(* CoDeSys 2.3.9.47 project: 1floor_2016_06_22_beta.pr6 *)
(* Libraries: TcBABasicBC.lb6 22.7.15 15:46:36, TcPlcUtilitiesBC.lb6 13.5.05 11:19:40, PlcSystemBC.lb6 21.3.01 11:03:02, TcAdsBC.lb6 5.7.02 11:03:02, standard.lb6 5.6.98 11:03:02 *)

(* Global variable list: main *)
VAR_GLOBAL


(*ADS*)

	ads_adr1: STRING:='10.0.5.61.1.1';
	ads_adr2: STRING:='10.0.5.62.1.1';
	ads_adr3: STRING:='10.0.5.63.1.1';

	write_ads: ADSWRITE;

	data2floor: ARRAY[0..3] OF BYTE;
	data2floor_prev :ARRAY[0..3] OF BYTE;
	data3floor: ARRAY[0..10] OF BYTE;
	data3floor_prev :ARRAY[0..10] OF BYTE;

	m_fancoil_vitalnya_low 			AT%MX300.0: BOOL;
	m_fancoil_vitalnya_med 			AT%MX300.1: BOOL;
	m_fancoil_vitalnya_high 			AT%MX300.2: BOOL;
	skvazhyna 						AT%MX300.3:BOOL;
	tepla_pidloga					AT%MX300.4:BOOL;

	T_out3							AT%MB303:BYTE;


	iHour							AT%MB304:BYTE;
	iMinute							AT%MB305:BYTE;
	lights							AT%MB306:DWORD;

	sw_tambur2_1					AT%MX200.0:BOOL;
	sw_tambur3_2					AT%MX300.1:BOOL;
	bDarkOutside					AT%MX300.6:BOOL;
	bT_out_sign						AT%MX300.7:BOOL;

	eib_komora_l 					AT%MX400.0:BOOL;
	eib_su1_l 						AT%MX400.1:BOOL;
	eib_topochna_l 					AT%MX400.2:BOOL;
	eib_su2_bra	 					AT%MX400.3:BOOL;
	eib_su2_l 						AT%MX400.4:BOOL;
	eib_su1_rakovyna 				AT%MX400.5:BOOL;
	eib_su2_dush 					AT%MX400.6:BOOL;
	eib_dush 						AT%MX400.7:BOOL;

	eib_kuhnya1	 				AT%MX401.0:BOOL;
	eib_vitalnya_smugy1 			AT%MX401.1:BOOL;
	eib_vitalnya_l 					AT%MX401.2:BOOL;
	eib_vitalnya_prokladka 			AT%MX401.3:BOOL;
	eib_terassa_stina	 			AT%MX401.4:BOOL;
	eib_pidval_shody	 			AT%MX401.5:BOOL;
	eib_skhody2pov 				AT%MX401.6:BOOL;
	eib_tambur_l 					AT%MX401.7:BOOL;

	eib_vent_su1 					AT%MX402.0:BOOL;
	eib_vent_kuh_low 				AT%MX402.1:BOOL;
	eib_vent_dush 					AT%MX402.2:BOOL;
	eib_vent_komora 				AT%MX402.3:BOOL;
	eib_vent_kuh_high 				AT%MX403.4:BOOL;

END_VAR

(* Global variable list: physical *)
VAR_GLOBAL



	moove_su1				AT %IX80.0:	BOOL;
	moove_topochna			AT %IX80.1:	BOOL;
	moove_su2				AT %IX80.2:	BOOL;
	moove_korydor_ops		AT %IX80.3:	BOOL;
	moove_korydor			AT %IX80.4:	BOOL;
	moove_vitalnya			AT %IX80.5:	BOOL;
	moove_komora			AT %IX80.6:	BOOL;
(*	din1_8	AT %IX80.7:	BOOL;*)
	moove_kino				AT %IX81.0:	BOOL;
	moove_skhody2_3		AT %IX81.1:	BOOL;
	moove_skhody1_2		AT %IX81.2:	BOOL;
	moove_garderob			AT %IX81.3:	BOOL;
	moove_studio			AT %IX81.4:	BOOL;
	moove_tambur3			AT %IX81.5:	BOOL;
	moove_kabinet			AT %IX81.6:	BOOL;
	moove_dytjacha			AT %IX81.7:	BOOL;
	moove_spalnya			AT %IX82.0:	BOOL;
(*	din3_2	AT %IX82.1:	BOOL;*)
	moove_korydor3			AT %IX82.2:	BOOL;
(*	din3_4	AT %IX82.3:	BOOL;
	din3_5	AT %IX82.4:	BOOL;
	din3_6	AT %IX82.5:	BOOL;
	din3_7	AT %IX82.6:	BOOL;
	din3_8sw_vhid2		AT %IX82.7:	BOOL;
	din4_1	AT %IX83.0:	BOOL;
*)
	sw_su1_2				AT %IX83.1:	BOOL;
	sw_komora1				AT %IX83.2:	BOOL;
	sw_vhid1					AT %IX83.3:	BOOL;
	sw_topochna2			AT %IX83.4:	BOOL;
	sw_vhid2					AT %IX83.5:	BOOL;
	sw_topochna1			AT %IX83.6:	BOOL;
	sw_su1_1				AT %IX83.7:	BOOL;
	sw_tambur1_2			AT %IX84.0:	BOOL;
	sw_su2					AT %IX84.1:	BOOL;
	sw_kuh_su2				AT %IX84.2:	BOOL;
	sw_kuh3					AT %IX84.3:	BOOL;
(*	din5_5	AT %IX84.4:	BOOL;*)
	sw_kuh4					AT %IX84.5:	BOOL;
	sw_tambur1				AT %IX84.6:	BOOL;
	sw_vitalnya1				AT %IX84.7:	BOOL;
	sw_vitalnya2				AT %IX85.0:	BOOL;
	sw_kuh2					AT %IX85.1:	BOOL;
(*	din6_3	AT %IX85.2:	BOOL;*)
	sw_kuh1					AT %IX85.3:	BOOL;
	sw_vitalnya3				AT %IX85.4:	BOOL;
	sw_tambur3				AT %IX85.5:	BOOL;
	sw_tambur_su			AT %IX85.6:	BOOL;
	sw_transit2pov			AT %IX85.7:	BOOL;

	ch_sensor1				AT %IX86.0:	BOOL;
	ch_sensor2				AT %IX86.1:	BOOL;
	zatoplennya_kot			AT %IX86.2:	BOOL;
	zatoplennya_komora		AT %IX86.3:	BOOL;
	zatoplennya_su2			AT %IX86.4:	BOOL;
	zatoplennya_kuh			AT %IX86.5:	BOOL;
	zatoplennya_su3pov		AT %IX86.6:	BOOL;
(*	din7_8	AT %IX86.7:	BOOL;*)

	komora_l				AT %QX80.0:	BOOL;
	su1_l					AT %QX80.1:	BOOL;
	topochna_l				AT %QX80.2:	BOOL;
	su2_bra					AT %QX80.3:	BOOL;
	topochna2_l				AT %QX80.4:	BOOL;
	su2_l					AT %QX80.5:	BOOL;
	su1_rakovyna			AT %QX80.6:	BOOL;
	su2_dush				AT %QX80.7:	BOOL;
	dush					AT %QX81.0:	BOOL;
	vitalnya_smugy2			AT %QX81.1:	BOOL;
	su2_polytsi				AT %QX81.2:	BOOL;
	fancoil_vitalnya_low		AT %QX81.3:	BOOL;
	kuhnya1					AT %QX81.4:	BOOL;
	fancoil_vitalnya_med		AT %QX81.5:	BOOL;
	kuhnya2					AT %QX81.6:	BOOL;
	fancoil_vitalnya_high		AT %QX81.7:	BOOL;
	w_valve_recirc			AT %QX82.0:	BOOL;
(*	dout3_2	AT %QX82.1:	BOOL;*)
	w_valve3pov				AT %QX82.2:	BOOL;
	vitalnya_smugy1			AT %QX82.3:	BOOL;
	w_valve1pov				AT %QX82.4:	BOOL;
	vitalnya_l				AT %QX82.5:	BOOL;
	freecooling				AT %QX82.6:	BOOL;
	vitalnya_prokladka		AT %QX82.7:	BOOL;
	terassa_stina				AT %QX83.0:	BOOL;
	pidval_shody				AT %QX83.1:	BOOL;
	terassa					AT %QX83.2:	BOOL;
	skhody2pov				AT %QX83.3:	BOOL;
(*	dout4_5	AT %QX83.4:	BOOL;
	dout4_6	AT %QX83.5:	BOOL;
*)	dout4_7	AT %QX83.6:	BOOL;

	tambur_l					AT %QX83.7:	BOOL;
(*	dout5_1	AT %QX84.0:	BOOL;
	dout5_2 AT %QX84.1:	BOOL;
*)	gas_valve				AT %QX84.2:	BOOL;
(*	dout5_4	AT %QX84.3:	BOOL;
	dout5_5	AT %QX84.4:	BOOL;
	dout5_6	AT %QX84.5:	BOOL;
	dout5_7	AT %QX84.6:	BOOL;
	dout5_8	AT %QX84.7:	BOOL;
	dout6_1	AT %QX85.0:	BOOL;
	dout6_2	AT %QX85.1:	BOOL;
	dout6_3	AT %QX85.2:	BOOL;
	dout6_4	AT %QX85.3:	BOOL;
	dout6_5	AT %QX85.4:	BOOL;
	dout6_6	AT %QX85.5:	BOOL;
	dout6_7	AT %QX85.6:	BOOL;
	dout6_8	AT %QX85.7:	BOOL;
	dout7_1	AT %QX86.0:	BOOL;
	dout7_2	AT %QX86.1:	BOOL;
	dout7_3	AT %QX86.2:	BOOL;
	dout7_4	AT %QX86.3:	BOOL;
	dout7_5	AT %QX86.4:	BOOL;
	dout7_6	AT %QX86.5:	BOOL;
	dout7_7	AT %QX86.6:	BOOL;
	dout7_8	AT %QX86.7:	BOOL;
	dout8_1	AT %QX87.0:	BOOL;
	dout8_2	AT %QX87.1:	BOOL;
	dout8_3	AT %QX87.2:	BOOL;
	dout8_4	AT %QX87.3:	BOOL;
	dout8_5	AT %QX87.4:	BOOL;
	dout8_6	AT %QX87.5:	BOOL;
	dout8_7	AT %QX87.6:	BOOL;
	dout8_8	AT %QX87.7:	BOOL;
*)	vent_su1					AT %QX88.0:	BOOL;
	vent_kuh_low				AT %QX88.1:	BOOL;
	vent_dush				AT %QX88.2:	BOOL;
	collector_komora			AT %QX88.3:	BOOL;
	vent_komora				AT %QX88.4:	BOOL;
	collector_kuh				AT %QX88.5:	BOOL;
	vent_kuh_high			AT %QX88.6:	BOOL;
	collector_vitalnya1			AT %QX88.7:	BOOL;
	collector_vitalnya2			AT %QX89.0:	BOOL;
(*	dout10_2	AT %QX89.1:	BOOL;
*)	collector_su2				AT %QX89.2:	BOOL;
(*	dout10_4	AT %QX89.3:	BOOL;
*)	collector_vhid_stina		AT %QX89.4:	BOOL;
(*	dout10_6	AT %QX89.5:	BOOL;
*)	collector_vhid				AT %QX89.6:	BOOL;
(*	dout10_8	AT %QX89.7:	BOOL;
	dout11_1	AT %QX90.0:	BOOL;
	dout11_2	AT %QX90.1:	BOOL;
	dout11_3	AT %QX90.2:	BOOL;
	dout11_4	AT %QX90.3:	BOOL;
	dout11_5	AT %QX90.4:	BOOL;
	dout11_6	AT %QX90.5:	BOOL;
	dout11_7	AT %QX90.6:	BOOL;
	dout11_8	AT %QX90.7:	BOOL;
*)
	klapan_vitalnya			AT %QB2:	INT;
	KL4414_2_Out			AT %QB6:	INT;
	KL4414_3_Out			AT %QB10:	INT;
	KL4414_4_Out			AT %QB14:	INT;

	temp_vhid	AT %IB50:	INT; (*25*)
	temp_dush	AT %IB58:	INT;(*25*)
	temp_kuh	AT %IB66:	INT;(*-136*)
	temp_vhid_stina	AT %IB70:	INT;(*0*)
(*
(* @GLOBAL_VARIABLE_LIST := TwinCAT_Import *)
(* @PATH := '' *)
VAR_GLOBAL (* DO NOT CHANGE THIS SHEET MANUALLY! *)
	PlcInVar_0	AT %QB128:	USINT;
	PlcInVar_1	AT %QB129:	USINT;
	PlcInVar_2	AT %QB130:	USINT;
	PlcInVar_3	AT %QB131:	USINT;
	PlcInVar_4	AT %QB132:	USINT;
	PlcInVar_5	AT %QB133:	USINT;
	PlcInVar_6	AT %QB134:	USINT;
	PlcInVar_7	AT %QB135:	USINT;
	PlcInVar_8	AT %QB136:	USINT;
	PlcInVar_9	AT %QB137:	USINT;
	PlcInVar_10	AT %QB138:	USINT;
	PlcInVar_11	AT %QB139:	USINT;
	PlcInVar_12	AT %QB140:	USINT;
	PlcInVar_13	AT %QB141:	USINT;
	PlcInVar_14	AT %QB142:	USINT;
	PlcInVar_15	AT %QB143:	USINT;
	PlcOutVar_0	AT %IB128:	USINT;
	PlcOutVar_1	AT %IB129:	USINT;
	PlcOutVar_2	AT %IB130:	USINT;
	PlcOutVar_3	AT %IB131:	USINT;
	PlcOutVar_4	AT %IB132:	USINT;
	PlcOutVar_5	AT %IB133:	USINT;
	PlcOutVar_6	AT %IB134:	USINT;
	PlcOutVar_7	AT %IB135:	USINT;
	PlcOutVar_8	AT %IB136:	USINT;
	PlcOutVar_9	AT %IB137:	USINT;
	PlcOutVar_10	AT %IB138:	USINT;
	PlcOutVar_11	AT %IB139:	USINT;
	PlcOutVar_12	AT %IB140:	USINT;
	PlcOutVar_13	AT %IB141:	USINT;
	PlcOutVar_14	AT %IB142:	USINT;
	PlcOutVar_15	AT %IB143:	USINT;
	Term_2_KL4414_1_State	AT %IB0:	USINT;
	Term_2_KL4414_1_Data_In	AT %IB2:	INT;
	Term_2_KL4414_1_Ctrl	AT %QB0:	USINT;
	Term_2_KL4414_1_Data_Out	AT %QB2:	INT;
	Term_2_KL4414_2_State	AT %IB4:	USINT;
	Term_2_KL4414_2_Data_In	AT %IB6:	INT;
	Term_2_KL4414_2_Ctrl	AT %QB4:	USINT;
	Term_2_KL4414_2_Data_Out	AT %QB6:	INT;
	Term_2_KL4414_3_State	AT %IB8:	USINT;
	Term_2_KL4414_3_Data_In	AT %IB10:	INT;
	Term_2_KL4414_3_Ctrl	AT %QB8:	USINT;
	Term_2_KL4414_3_Data_Out	AT %QB10:	INT;
	Term_2_KL4414_4_State	AT %IB12:	USINT;
	Term_2_KL4414_4_Data_In	AT %IB14:	INT;
	Term_2_KL4414_4_Ctrl	AT %QB12:	USINT;
	Term_2_KL4414_4_Data_Out	AT %QB14:	INT;
	Term_14_KL3228_4_1_State	AT %IB16:	USINT;
	Term_14_KL3228_4_1_Data_In	AT %IB18:	INT;
	Term_14_KL3228_4_1_Ctrl	AT %QB16:	USINT;
	Term_14_KL3228_4_1_Data_Out	AT %QB18:	INT;
	Term_14_KL3228_4_2_State	AT %IB20:	USINT;
	Term_14_KL3228_4_2_Data_In	AT %IB22:	INT;
	Term_14_KL3228_4_2_Ctrl	AT %QB20:	USINT;
	Term_14_KL3228_4_2_Data_Out	AT %QB22:	INT;
	Term_14_KL3228_4_3_State	AT %IB24:	USINT;
	Term_14_KL3228_4_3_Data_In	AT %IB26:	INT;
	Term_14_KL3228_4_3_Ctrl	AT %QB24:	USINT;
	Term_14_KL3228_4_3_Data_Out	AT %QB26:	INT;
	Term_14_KL3228_4_4_State	AT %IB28:	USINT;
	Term_14_KL3228_4_4_Data_In	AT %IB30:	INT;
	Term_14_KL3228_4_4_Ctrl	AT %QB28:	USINT;
	Term_14_KL3228_4_4_Data_Out	AT %QB30:	INT;
	Term_15_KL3228_4_1_State	AT %IB32:	USINT;
	Term_15_KL3228_4_1_Data_In	AT %IB34:	INT;
	Term_15_KL3228_4_1_Ctrl	AT %QB32:	USINT;
	Term_15_KL3228_4_1_Data_Out	AT %QB34:	INT;
	Term_15_KL3228_4_2_State	AT %IB36:	USINT;
	Term_15_KL3228_4_2_Data_In	AT %IB38:	INT;
	Term_15_KL3228_4_2_Ctrl	AT %QB36:	USINT;
	Term_15_KL3228_4_2_Data_Out	AT %QB38:	INT;
	Term_15_KL3228_4_3_State	AT %IB40:	USINT;
	Term_15_KL3228_4_3_Data_In	AT %IB42:	INT;
	Term_15_KL3228_4_3_Ctrl	AT %QB40:	USINT;
	Term_15_KL3228_4_3_Data_Out	AT %QB42:	INT;
	Term_15_KL3228_4_4_State	AT %IB44:	USINT;
	Term_15_KL3228_4_4_Data_In	AT %IB46:	INT;
	Term_15_KL3228_4_4_Ctrl	AT %QB44:	USINT;
	Term_15_KL3228_4_4_Data_Out	AT %QB46:	INT;
	Term_16_KL3228_4_1_State	AT %IB48:	USINT;
	Term_16_KL3228_4_1_Data_In	AT %IB50:	INT;
	Term_16_KL3228_4_1_Ctrl	AT %QB48:	USINT;
	Term_16_KL3228_4_1_Data_Out	AT %QB50:	INT;
	Term_16_KL3228_4_2_State	AT %IB52:	USINT;
	Term_16_KL3228_4_2_Data_In	AT %IB54:	INT;
	Term_16_KL3228_4_2_Ctrl	AT %QB52:	USINT;
	Term_16_KL3228_4_2_Data_Out	AT %QB54:	INT;
	Term_16_KL3228_4_3_State	AT %IB56:	USINT;
	Term_16_KL3228_4_3_Data_In	AT %IB58:	INT;
	Term_16_KL3228_4_3_Ctrl	AT %QB56:	USINT;
	Term_16_KL3228_4_3_Data_Out	AT %QB58:	INT;
	Term_16_KL3228_4_4_State	AT %IB60:	USINT;
	Term_16_KL3228_4_4_Data_In	AT %IB62:	INT;
	Term_16_KL3228_4_4_Ctrl	AT %QB60:	USINT;
	Term_16_KL3228_4_4_Data_Out	AT %QB62:	INT;
	Term_17_KL3228_4_1_State	AT %IB64:	USINT;
	Term_17_KL3228_4_1_Data_In	AT %IB66:	INT;
	Term_17_KL3228_4_1_Ctrl	AT %QB64:	USINT;
	Term_17_KL3228_4_1_Data_Out	AT %QB66:	INT;
	Term_17_KL3228_4_2_State	AT %IB68:	USINT;
	Term_17_KL3228_4_2_Data_In	AT %IB70:	INT;
	Term_17_KL3228_4_2_Ctrl	AT %QB68:	USINT;
	Term_17_KL3228_4_2_Data_Out	AT %QB70:	INT;
	Term_17_KL3228_4_3_State	AT %IB72:	USINT;
	Term_17_KL3228_4_3_Data_In	AT %IB74:	INT;
	Term_17_KL3228_4_3_Ctrl	AT %QB72:	USINT;
	Term_17_KL3228_4_3_Data_Out	AT %QB74:	INT;
	Term_17_KL3228_4_4_State	AT %IB76:	USINT;
	Term_17_KL3228_4_4_Data_In	AT %IB78:	INT;
	Term_17_KL3228_4_4_Ctrl	AT %QB76:	USINT;
	Term_17_KL3228_4_4_Data_Out	AT %QB78:	INT; 
	Term_3_KL2408_1_Output	AT %QX80.0:	BOOL;
	Term_3_KL2408_2_Output	AT %QX80.1:	BOOL;
	Term_3_KL2408_3_Output	AT %QX80.2:	BOOL;
	Term_3_KL2408_4_Output	AT %QX80.3:	BOOL;
	Term_3_KL2408_5_Output	AT %QX80.4:	BOOL;
	Term_3_KL2408_6_Output	AT %QX80.5:	BOOL;
	Term_3_KL2408_7_Output	AT %QX80.6:	BOOL;
	Term_3_KL2408_8_Output	AT %QX80.7:	BOOL;
	Term_4_KL2408_1_Output	AT %QX81.0:	BOOL;
	Term_4_KL2408_2_Output	AT %QX81.1:	BOOL;
	Term_4_KL2408_3_Output	AT %QX81.2:	BOOL;
	Term_4_KL2408_4_Output	AT %QX81.3:	BOOL;
	Term_4_KL2408_5_Output	AT %QX81.4:	BOOL;
	Term_4_KL2408_6_Output	AT %QX81.5:	BOOL;
	Term_4_KL2408_7_Output	AT %QX81.6:	BOOL;
	Term_4_KL2408_8_Output	AT %QX81.7:	BOOL;
	Term_5_KL2408_1_Output	AT %QX82.0:	BOOL;
	Term_5_KL2408_2_Output	AT %QX82.1:	BOOL;
	Term_5_KL2408_3_Output	AT %QX82.2:	BOOL;
	Term_5_KL2408_4_Output	AT %QX82.3:	BOOL;
	Term_5_KL2408_5_Output	AT %QX82.4:	BOOL;
	Term_5_KL2408_6_Output	AT %QX82.5:	BOOL;
	Term_5_KL2408_7_Output	AT %QX82.6:	BOOL;
	Term_5_KL2408_8_Output	AT %QX82.7:	BOOL;
	Term_6_KL2408_1_Output	AT %QX83.0:	BOOL;
	Term_6_KL2408_2_Output	AT %QX83.1:	BOOL;
	Term_6_KL2408_3_Output	AT %QX83.2:	BOOL;
	Term_6_KL2408_4_Output	AT %QX83.3:	BOOL;
	Term_6_KL2408_5_Output	AT %QX83.4:	BOOL;
	Term_6_KL2408_6_Output	AT %QX83.5:	BOOL;
	Term_6_KL2408_7_Output	AT %QX83.6:	BOOL;
	Term_6_KL2408_8_Output	AT %QX83.7:	BOOL;
	Term_7_KL2408_1_Output	AT %QX84.0:	BOOL;
	Term_7_KL2408_2_Output	AT %QX84.1:	BOOL;
	Term_7_KL2408_3_Output	AT %QX84.2:	BOOL;
	Term_7_KL2408_4_Output	AT %QX84.3:	BOOL;
	Term_7_KL2408_5_Output	AT %QX84.4:	BOOL;
	Term_7_KL2408_6_Output	AT %QX84.5:	BOOL;
	Term_7_KL2408_7_Output	AT %QX84.6:	BOOL;
	Term_7_KL2408_8_Output	AT %QX84.7:	BOOL;
	Term_8_KL2408_1_Output	AT %QX85.0:	BOOL;
	Term_8_KL2408_2_Output	AT %QX85.1:	BOOL;
	Term_8_KL2408_3_Output	AT %QX85.2:	BOOL;
	Term_8_KL2408_4_Output	AT %QX85.3:	BOOL;
	Term_8_KL2408_5_Output	AT %QX85.4:	BOOL;
	Term_8_KL2408_6_Output	AT %QX85.5:	BOOL;
	Term_8_KL2408_7_Output	AT %QX85.6:	BOOL;
	Term_8_KL2408_8_Output	AT %QX85.7:	BOOL;
	Term_9_KL2408_1_Output	AT %QX86.0:	BOOL;
	Term_9_KL2408_2_Output	AT %QX86.1:	BOOL;
	Term_9_KL2408_3_Output	AT %QX86.2:	BOOL;
	Term_9_KL2408_4_Output	AT %QX86.3:	BOOL;
	Term_9_KL2408_5_Output	AT %QX86.4:	BOOL;
	Term_9_KL2408_6_Output	AT %QX86.5:	BOOL;
	Term_9_KL2408_7_Output	AT %QX86.6:	BOOL;
	Term_9_KL2408_8_Output	AT %QX86.7:	BOOL;
	Term_10_KL2408_1_Output	AT %QX87.0:	BOOL;
	Term_10_KL2408_2_Output	AT %QX87.1:	BOOL;
	Term_10_KL2408_3_Output	AT %QX87.2:	BOOL;
	Term_10_KL2408_4_Output	AT %QX87.3:	BOOL;
	Term_10_KL2408_5_Output	AT %QX87.4:	BOOL;
	Term_10_KL2408_6_Output	AT %QX87.5:	BOOL;
	Term_10_KL2408_7_Output	AT %QX87.6:	BOOL;
	Term_10_KL2408_8_Output	AT %QX87.7:	BOOL;
	Term_11_KL2408_1_Output	AT %QX88.0:	BOOL;
	Term_11_KL2408_2_Output	AT %QX88.1:	BOOL;
	Term_11_KL2408_3_Output	AT %QX88.2:	BOOL;
	Term_11_KL2408_4_Output	AT %QX88.3:	BOOL;
	Term_11_KL2408_5_Output	AT %QX88.4:	BOOL;
	Term_11_KL2408_6_Output	AT %QX88.5:	BOOL;
	Term_11_KL2408_7_Output	AT %QX88.6:	BOOL;
	Term_11_KL2408_8_Output	AT %QX88.7:	BOOL;
	Term_12_KL2408_1_Output	AT %QX89.0:	BOOL;
	Term_12_KL2408_2_Output	AT %QX89.1:	BOOL;
	Term_12_KL2408_3_Output	AT %QX89.2:	BOOL;
	Term_12_KL2408_4_Output	AT %QX89.3:	BOOL;
	Term_12_KL2408_5_Output	AT %QX89.4:	BOOL;
	Term_12_KL2408_6_Output	AT %QX89.5:	BOOL;
	Term_12_KL2408_7_Output	AT %QX89.6:	BOOL;
	Term_12_KL2408_8_Output	AT %QX89.7:	BOOL;
	Term_13_KL2408_1_Output	AT %QX90.0:	BOOL;
	Term_13_KL2408_2_Output	AT %QX90.1:	BOOL;
	Term_13_KL2408_3_Output	AT %QX90.2:	BOOL;
	Term_13_KL2408_4_Output	AT %QX90.3:	BOOL;
	Term_13_KL2408_5_Output	AT %QX90.4:	BOOL;
	Term_13_KL2408_6_Output	AT %QX90.5:	BOOL;
	Term_13_KL2408_7_Output	AT %QX90.6:	BOOL;
	Term_13_KL2408_8_Output	AT %QX90.7:	BOOL;
	
END_VAR

*)
END_VAR

(* Data type *)
TYPE ContactType: (NO,NC);
(*NO - sensor sends TRUE on triggering and FALSE in normal state.
NC - sensor sends FALSE on triggering and TRUE in normal state *)

END_TYPE

(* Data type *)
TYPE   ManSwitch: (OFF, ON, AUTO);
END_TYPE

(* Data type *)
TYPE ROOM_HVAC :
STRUCT

	heat_mode:STRING;
	heat_speed:USINT;

	delta_t:SINT;
	t_cur:SINT;
	t_ust:SINT;

	fancoil_speed:SINT;
	klapan:WORD;

	collector1: BOOL;
	collector2: BOOL;
	collector3: BOOL;
	collector4: BOOL;

END_STRUCT
END_TYPE

(* Data type *)
TYPE WaterLeakageDetectionCfg :
	STRUCT
		sensorContacts:ContactType:=NO;
		valveContacts:ContactType:=NO;
		sensorDelay:TIME:=t#5s;
		waterOnTimerDelay: TIME:=t#10ms;
	END_STRUCT
END_TYPE

(* POU MAIN, ST *)
PROGRAM MAIN
VAR

	i:INT;
END_VAR
WaterAndGasLeakage;
Light;
heat;
ADS_write;
END_PROGRAM

(* POU WaterAndGasLeakage, FBD *)
PROGRAM WaterAndGasLeakage
VAR
	defaultCfg: WaterLeakageDetectionCfg;
	gasValveCfg: WaterLeakageDetectionCfg:=(
		sensorContacts:=NC,
		valveContacts:=NO,
		sensorDelay:=t#5s,
		waterOnTimerDelay:=t#0ms
		);
	firstFloorLeakageDetection: fbWaterLeakage;
	thirdFloorLeakageDetection: fbWaterLeakage;
	tempReset: BOOL;
	firstFloorWaterAlarm, thirdFloorWaterAlarm:BOOL;
	firstFloorWaterState, thirdFloorWaterState:BOOL;

	gasAlarm: BOOL;
	gasState: BOOL;
END_VAR
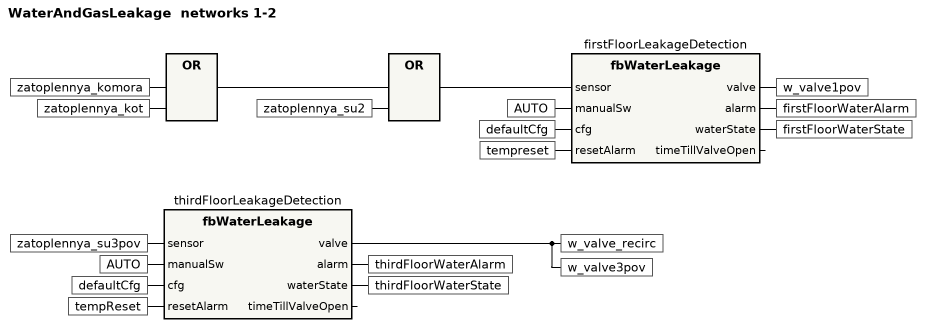
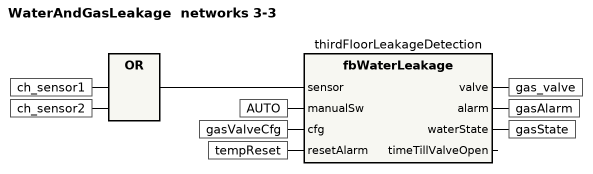
_FBD_ (* Function Block Diagram *)
NETWORK 1
	firstFloorLeakageDetection:fbWaterLeakage(sensor: OR(OR(zatoplennya_komora, zatoplennya_kot), zatoplennya_su2), manualSw: AUTO, cfg: defaultCfg, resetAlarm: tempreset, alarm => firstFloorWaterAlarm, waterState => firstFloorWaterState) => w_valve1pov
NETWORK 2
	thirdFloorLeakageDetection:fbWaterLeakage(sensor: zatoplennya_su3pov, manualSw: AUTO, cfg: defaultCfg, resetAlarm: tempReset, alarm => thirdFloorWaterAlarm, waterState => thirdFloorWaterState) => w_valve_recirc, w_valve3pov
NETWORK 3
	thirdFloorLeakageDetection:fbWaterLeakage(sensor: OR(ch_sensor1, ch_sensor2), manualSw: AUTO, cfg: gasValveCfg, resetAlarm: tempReset, alarm => gasAlarm, waterState => gasState) => gas_valve
_END_FBD_
(* the same logic as Structured Text *)
(* Network 1 *)
firstFloorLeakageDetection(sensor := (zatoplennya_komora OR zatoplennya_kot) OR zatoplennya_su2, manualSw := AUTO, cfg := defaultCfg, resetAlarm := tempreset);
firstFloorWaterAlarm := firstFloorLeakageDetection.alarm;
firstFloorWaterState := firstFloorLeakageDetection.waterState;
w_valve1pov := firstFloorLeakageDetection.valve;
(* Network 2 *)
thirdFloorLeakageDetection(sensor := zatoplennya_su3pov, manualSw := AUTO, cfg := defaultCfg, resetAlarm := tempReset);
thirdFloorWaterAlarm := thirdFloorLeakageDetection.alarm;
thirdFloorWaterState := thirdFloorLeakageDetection.waterState;
w_valve_recirc := thirdFloorLeakageDetection.valve;
w_valve3pov := thirdFloorLeakageDetection.valve;
(* Network 3 *)
thirdFloorLeakageDetection(sensor := ch_sensor1 OR ch_sensor2, manualSw := AUTO, cfg := gasValveCfg, resetAlarm := tempReset);
gasAlarm := thirdFloorLeakageDetection.alarm;
gasState := thirdFloorLeakageDetection.waterState;
gas_valve := thirdFloorLeakageDetection.valve;
END_PROGRAM

(* POU fbWaterLeakage, ST *)
FUNCTION_BLOCK fbWaterLeakage
VAR_INPUT
	sensor:BOOL;
 	manualSw				: ManSwitch;              (*button in UI FOR manual mode switching*)
END_VAR
VAR_OUTPUT
	valve					: BOOL;                      (*hardware output*)
	alarm					: BOOL	:=FALSE;
	waterState				: BOOL;			 (*shows IF valve is open*)
	timeTillValveOpen			: TIME;			(*informational output FOR user TO know in how much TIME water will turn on*)
END_VAR

VAR_IN_OUT
            cfg						:  WaterLeakageDetectionCfg;
            resetAlarm				: BOOL;

  END_VAR

VAR
 	alarmSet					: SR;			(*Sets alarm in CASE OF water leakage AND resets it on "resetAlarm" going TRUE*)
	sensorLagTimer 			: TON;
	waterOnAfterAlarmTimer	: TON;       		(*Makes a delay after alarm was reseted AND before turning on water*)
END_VAR
  (*
  manual mode switching.
  ON - valve is permanently open,
  OFF - valve is permanently closed,
  AUTO - vale position is  controled by fb logic
  *)
  CASE manualSw OF
  
       AUTO:
            (*setting alarm on if sensor is still in alarm state ater delay*)
            sensorLagTimer.PT:=cfg.sensorDelay;
            CASE cfg.sensorContacts OF
                 NC:
                    sensorLagTimer(IN :=NOT sensor);
                    alarmSet.SET1:=NOT sensor AND sensorLagTimer.Q;
                 NO:
                    sensorLagTimer(IN := sensor);
                    alarmSet.SET1:= sensor AND sensorLagTimer.Q;
            END_CASE;

            alarmSet(RESET:=resetAlarm AND waterOnAfterAlarmTimer.Q, q1=>alarm);


            waterOnAfterAlarmTimer(IN :=(alarm AND resetAlarm), PT:=cfg.waterOnTimerDelay);


            (*switching water on after alarm with a delay*)
            waterState:=  NOT alarm;

            IF NOT alarm THEN
                  waterState:=TRUE;
            ELSE
                waterState:=FALSE;
            END_IF;

            IF sensorLagTimer.ET<>t#0s OR waterState THEN       (*deactivating this input if there is a signal from sensor or when alarm goes off*)
               resetAlarm:=FALSE;                               (*This done to make it act like an impulse switch so user shouldn't deactivate "resetAlarm" manualy*)
            END_IF;

  ON:
       waterState:=TRUE;
  OFF:
       waterState:=FALSE;
  END_CASE;


  (*Set valve state depending on its config*)
  CASE cfg.valveContacts OF
     NC:
        valve:= waterState;
     NO:
        valve:=NOT waterState;
  END_CASE;

  (*calculating remaining time till water turns on*)
  timeTillValveOpen:=cfg.waterOnTimerDelay-waterOnAfterAlarmTimer.ET;
END_FUNCTION_BLOCK

(* POU lights/Light, CFC *)
PROGRAM Light
VAR
	longPressDelay: TIME:=t#500ms;
	lightDuration:TIME:=t#2m;



	fbSu1_l									: FB_Light;							(*fb for switching light group in wc near main enterance*)

	fbSu2_l									: FB_Light;							(*fb for switching main light group in wc with a shower*)
	fbSu2_bra								: FB_Light;							(*fb for switching bra group in wc with a shower*)
	fbSu1_rakovyna							: FB_Light;							(*fb for switching light group on the ceiling above washing basin in wc near main enterance*)
	fbSu2_dush								: FB_Light;							(*fb for light group in wc with a shower*)
	fbDush									: FB_Light;							(*fb for switching light in a shower room*)
	fbKuh_su2_sw							: FB_ShortLongClick;				(*process signals from switch in kitchen near shower#2 enterance*)
	fbDush_sw								: FB_ShortLongClick;				(*process signals from switch in su2 near the shower *)
	fbDush_vent							: FB_Light;							(*fb for shover fan switching*)
	fbSmugy								: FB_Light;							(*fb for switching LED stripes in livingroom*)
	fbKuhnya								: FB_Light;							(*fb for switching main lightgroup in "kitchen" part of the livingroom*)
	fbVitalnya_l								: FB_Light;							(*fb for switching main lightgroup in livinngroom*)
	fbProkladka								: FB_Light;							(*fb for switching curved LED lightgroup on the livingroom ceiling *)
	fbTerassa								: FB_Light;							(*fb for switching terrade lights in the floor *)
	fbTerassa_stina							: FB_Light;							(*fb for switching terrade lights on the wall*)
	fbTambur3_sw							: FB_ShortLongClick;				(*process signals from third switch in first floor hall*)
	fbPidval_shody							: FB_Light;							(*fb for switching light on stairs to the basement junction*)
	fbTamburFirstFloor						: FB_StairwellLight;					(*fb for switching 'zebra' light in first floor hall*)
	fbSkhody2Pov							: FB_Light;							(*fb for switching wall bras on the stairway to 2 floor*)
	fbKuhnyaVent							: FB_Light;							(*fb for switching fan in kitchen above the stove*)
	fbKuh1_sw								: FB_ShortLongClick;				(*process signals from switch near livingroom door*)
	fbSu1_1sw								: FB_ShortLongClick;				(*process signals from switch in WC near main entrance*)
	fbSu1Vent								: FB_Light;							(*fb for switching fan in WC near main enterance*)
	fbKomora1_sw							: FB_ShortLongClick;				(*processing signals from switch in tech room*)
	fbKomoraVent							: FB_Light;							(*fb for switching fan in tech room*)
	fbKomoraLight							: fbMoovingSensorLight;
	fbTopochnaLight						: fbMoovingSensorLight;
	fbTamburLight							: fbMoovingSensorLight;
END_VAR
VAR CONSTANT
	msecMultiplier: DINT := 1000;
END_VAR
VAR_OUTPUT

END_VAR
VAR (* helpers for the ST form of the networks *)
	_t691 : BOOL;
	_t520 : BOOL;
END_VAR
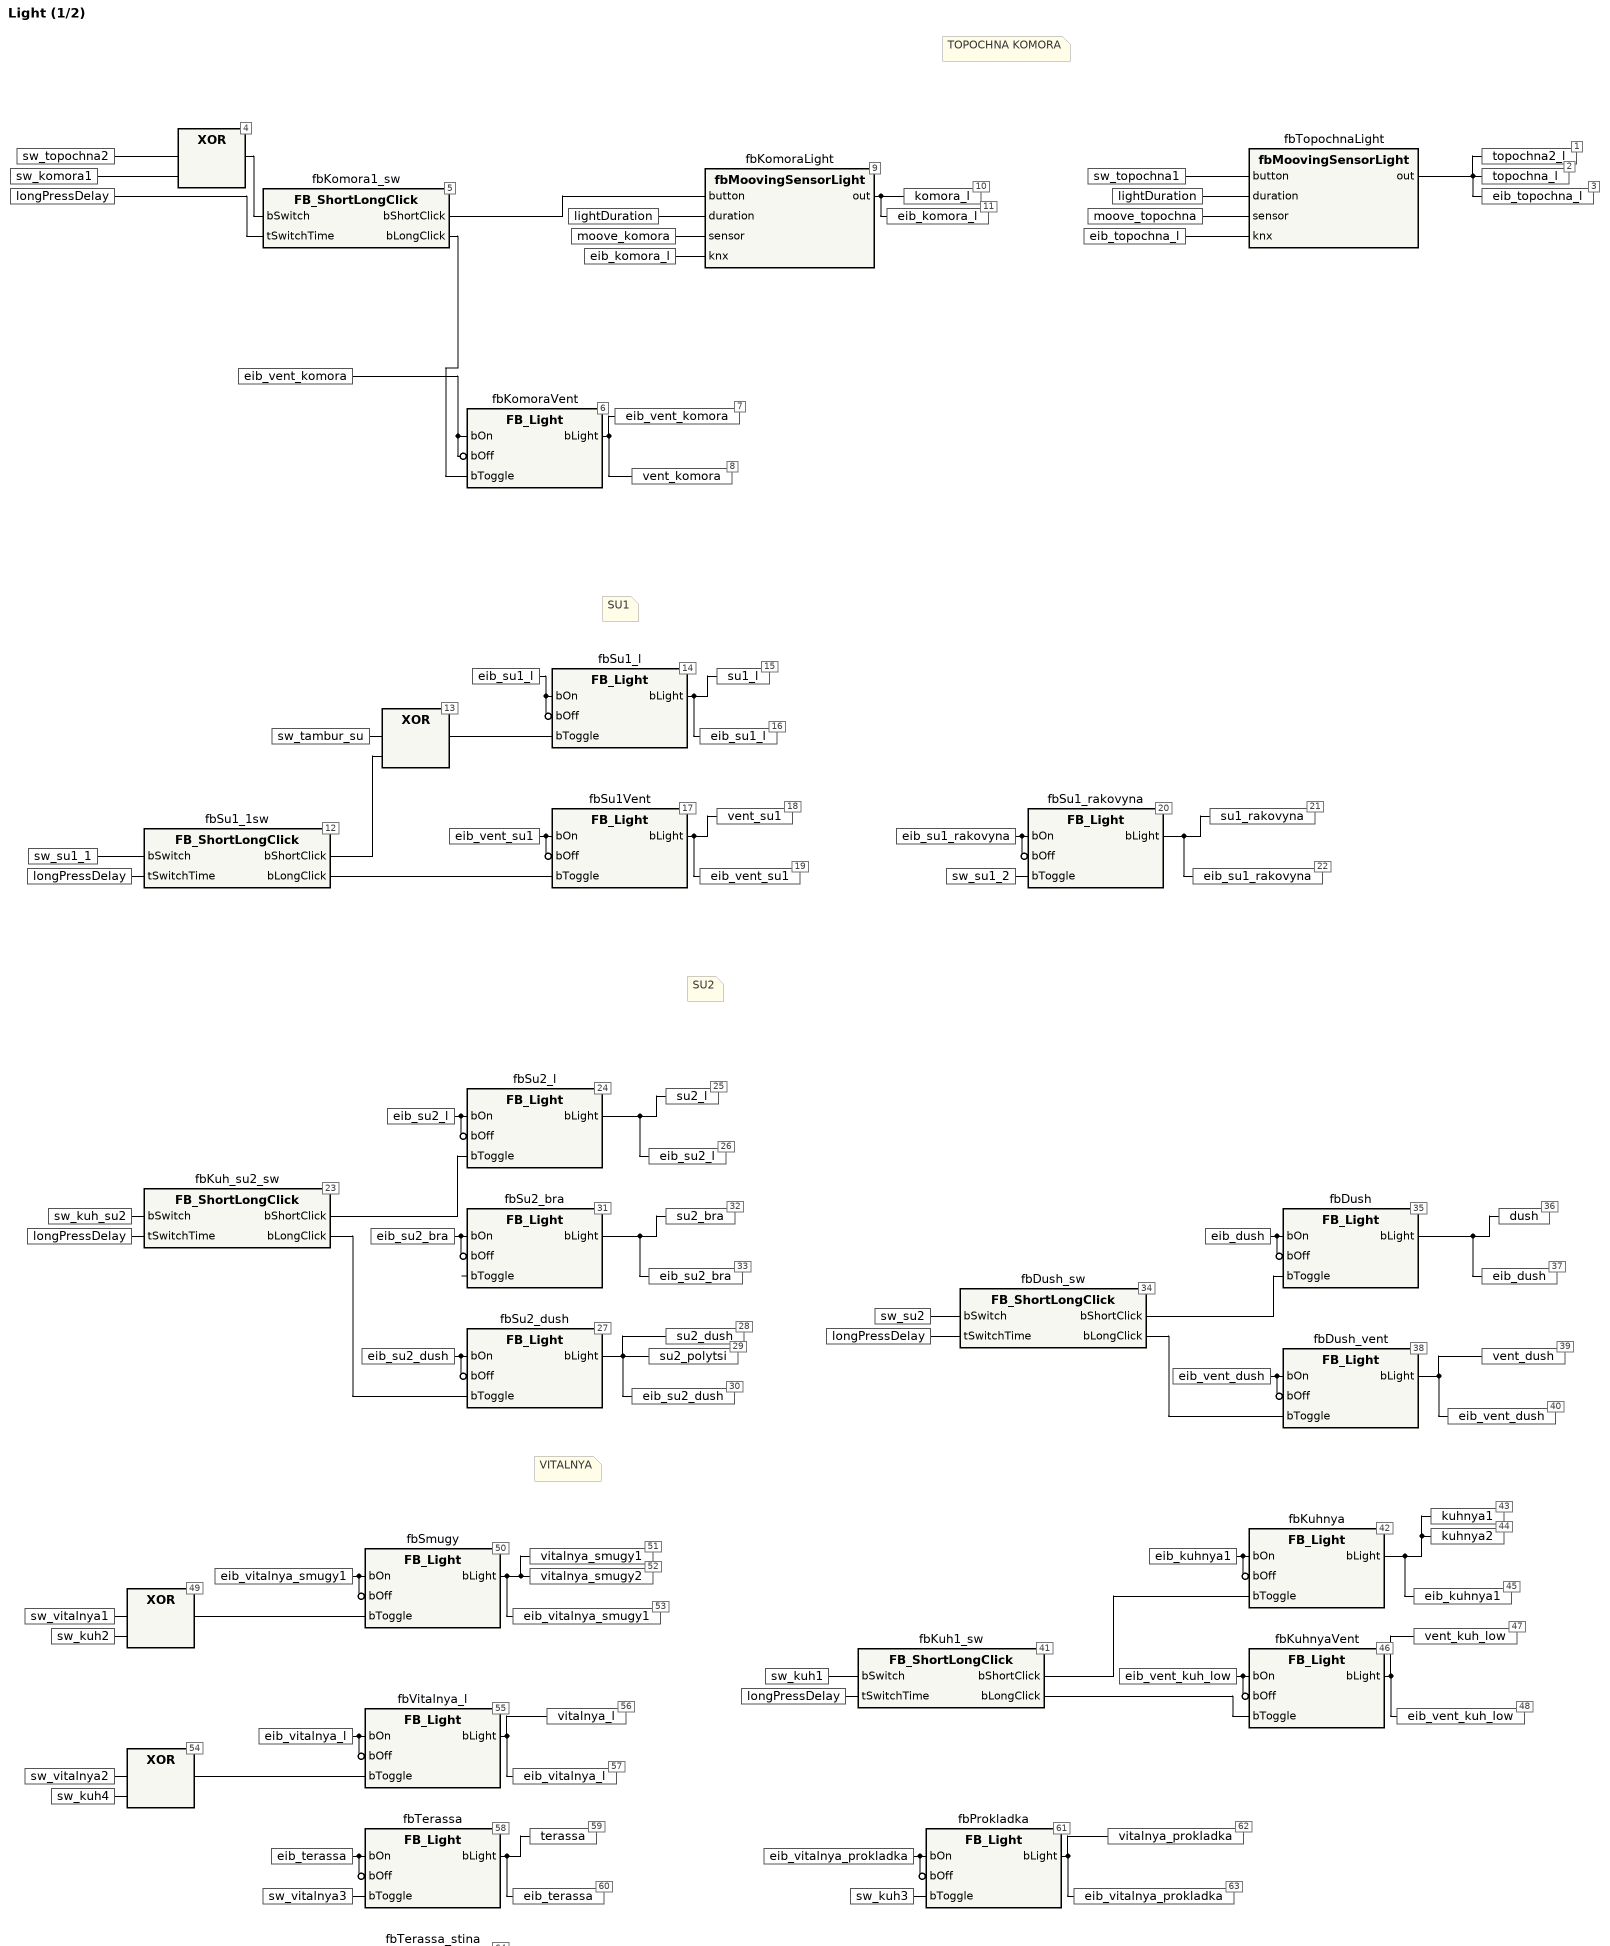
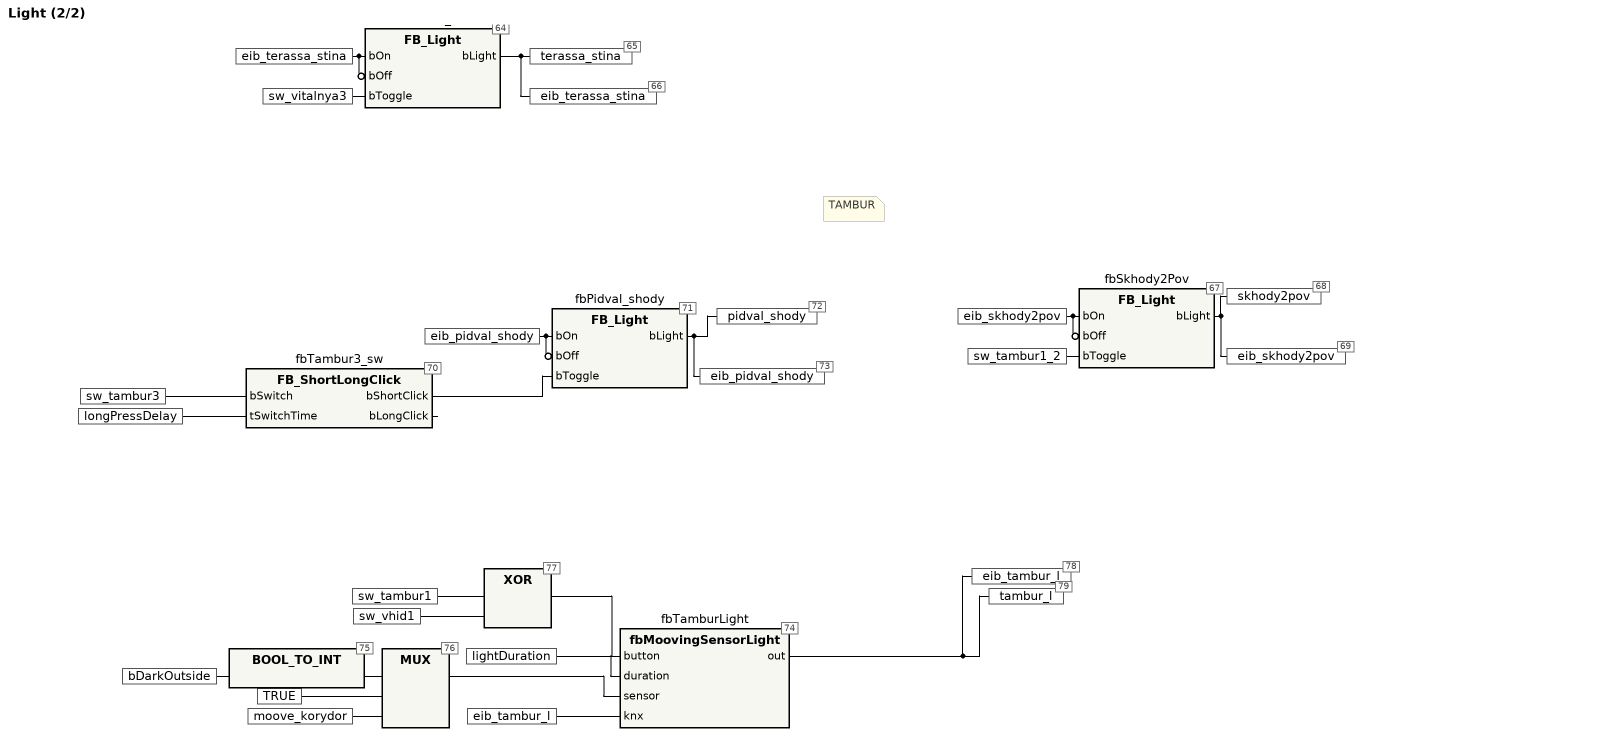
_CFC_ (* Continuous Function Chart, elements in execution order *)
(* TAMBUR *)
(* SU2 *)
(* VITALNYA *)
(* SU1 *)
(* TOPOCHNA KOMORA *)
#0 fbTopochnaLight:fbMoovingSensorLight(button: sw_topochna1, duration: lightDuration, sensor: moove_topochna, knx: eib_topochna_l)
#1 topochna2_l <= #0.out
#2 topochna_l <= #0.out
#3 eib_topochna_l <= #0.out
#4 XOR(sw_topochna2, sw_komora1)
#5 fbKomora1_sw:FB_ShortLongClick(bSwitch: #4, tSwitchTime: longPressDelay)
#6 fbKomoraVent:FB_Light(bOn: eib_vent_komora, bOff: NOT eib_vent_komora, bToggle: #5.bLongClick)
#7 eib_vent_komora <= #6.bLight
#8 vent_komora <= #6.bLight
#9 fbKomoraLight:fbMoovingSensorLight(button: #5.bShortClick, duration: lightDuration, sensor: moove_komora, knx: eib_komora_l)
#10 komora_l <= #9.out
#11 eib_komora_l <= #9.out
#12 fbSu1_1sw:FB_ShortLongClick(bSwitch: sw_su1_1, tSwitchTime: longPressDelay)
#13 XOR(sw_tambur_su, #12.bShortClick)
#14 fbSu1_l:FB_Light(bOn: eib_su1_l, bOff: NOT eib_su1_l, bToggle: #13)
#15 su1_l <= #14.bLight
#16 eib_su1_l <= #14.bLight
#17 fbSu1Vent:FB_Light(bOn: eib_vent_su1, bOff: NOT eib_vent_su1, bToggle: #12.bLongClick)
#18 vent_su1 <= #17.bLight
#19 eib_vent_su1 <= #17.bLight
#20 fbSu1_rakovyna:FB_Light(bOn: eib_su1_rakovyna, bOff: NOT eib_su1_rakovyna, bToggle: sw_su1_2)
#21 su1_rakovyna <= #20.bLight
#22 eib_su1_rakovyna <= #20.bLight
#23 fbKuh_su2_sw:FB_ShortLongClick(bSwitch: sw_kuh_su2, tSwitchTime: longPressDelay)
#24 fbSu2_l:FB_Light(bOn: eib_su2_l, bOff: NOT eib_su2_l, bToggle: #23.bShortClick)
#25 su2_l <= #24.bLight
#26 eib_su2_l <= #24.bLight
#27 fbSu2_dush:FB_Light(bOn: eib_su2_dush, bOff: NOT eib_su2_dush, bToggle: #23.bLongClick)
#28 su2_dush <= #27.bLight
#29 su2_polytsi <= #27.bLight
#30 eib_su2_dush <= #27.bLight
#31 fbSu2_bra:FB_Light(bOn: eib_su2_bra, bOff: NOT eib_su2_bra, bToggle: -)
#32 su2_bra <= #31.bLight
#33 eib_su2_bra <= #31.bLight
#34 fbDush_sw:FB_ShortLongClick(bSwitch: sw_su2, tSwitchTime: longPressDelay)
#35 fbDush:FB_Light(bOn: eib_dush, bOff: NOT eib_dush, bToggle: #34.bShortClick)
#36 dush <= #35.bLight
#37 eib_dush <= #35.bLight
#38 fbDush_vent:FB_Light(bOn: eib_vent_dush, bOff: NOT eib_vent_dush, bToggle: #34.bLongClick)
#39 vent_dush <= #38.bLight
#40 eib_vent_dush <= #38.bLight
#41 fbKuh1_sw:FB_ShortLongClick(bSwitch: sw_kuh1, tSwitchTime: longPressDelay)
#42 fbKuhnya:FB_Light(bOn: eib_kuhnya1, bOff: NOT eib_kuhnya1, bToggle: #41.bShortClick)
#43 kuhnya1 <= #42.bLight
#44 kuhnya2 <= #42.bLight
#45 eib_kuhnya1 <= #42.bLight
#46 fbKuhnyaVent:FB_Light(bOn: eib_vent_kuh_low, bOff: NOT eib_vent_kuh_low, bToggle: #41.bLongClick)
#47 vent_kuh_low <= #46.bLight
#48 eib_vent_kuh_low <= #46.bLight
#49 XOR(sw_vitalnya1, sw_kuh2)
#50 fbSmugy:FB_Light(bOn: eib_vitalnya_smugy1, bOff: NOT eib_vitalnya_smugy1, bToggle: #49)
#51 vitalnya_smugy1 <= #50.bLight
#52 vitalnya_smugy2 <= #50.bLight
#53 eib_vitalnya_smugy1 <= #50.bLight
#54 XOR(sw_vitalnya2, sw_kuh4)
#55 fbVitalnya_l:FB_Light(bOn: eib_vitalnya_l, bOff: NOT eib_vitalnya_l, bToggle: #54)
#56 vitalnya_l <= #55.bLight
#57 eib_vitalnya_l <= #55.bLight
#58 fbTerassa:FB_Light(bOn: eib_terassa, bOff: NOT eib_terassa, bToggle: sw_vitalnya3)
#59 terassa <= #58.bLight
#60 eib_terassa <= #58.bLight
#61 fbProkladka:FB_Light(bOn: eib_vitalnya_prokladka, bOff: NOT eib_vitalnya_prokladka, bToggle: sw_kuh3)
#62 vitalnya_prokladka <= #61.bLight
#63 eib_vitalnya_prokladka <= #61.bLight
#64 fbTerassa_stina:FB_Light(bOn: eib_terassa_stina, bOff: NOT eib_terassa_stina, bToggle: sw_vitalnya3)
#65 terassa_stina <= #64.bLight
#66 eib_terassa_stina <= #64.bLight
#67 fbSkhody2Pov:FB_Light(bOn: eib_skhody2pov, bOff: NOT eib_skhody2pov, bToggle: sw_tambur1_2)
#68 skhody2pov <= #67.bLight
#69 eib_skhody2pov <= #67.bLight
#70 fbTambur3_sw:FB_ShortLongClick(bSwitch: sw_tambur3, tSwitchTime: longPressDelay)
#71 fbPidval_shody:FB_Light(bOn: eib_pidval_shody, bOff: NOT eib_pidval_shody, bToggle: #70.bShortClick)
#72 pidval_shody <= #71.bLight
#73 eib_pidval_shody <= #71.bLight
#74 fbTamburLight:fbMoovingSensorLight(button: #77, duration: lightDuration, sensor: #76, knx: eib_tambur_l)
#75 BOOL_TO_INT(bDarkOutside)
#76 MUX(#75, TRUE, moove_korydor)
#77 XOR(sw_tambur1, sw_vhid1)
#78 eib_tambur_l <= #74.out
#79 tambur_l <= #74.out
_END_CFC_
(* the same logic as Structured Text *)
(* TAMBUR *)
(* SU2 *)
(* VITALNYA *)
(* SU1 *)
(* TOPOCHNA KOMORA *)
fbTopochnaLight(button := sw_topochna1, duration := lightDuration, sensor := moove_topochna, knx := eib_topochna_l);
topochna2_l := fbTopochnaLight.out;
topochna_l := fbTopochnaLight.out;
eib_topochna_l := fbTopochnaLight.out;
fbKomora1_sw(bSwitch := sw_topochna2 XOR sw_komora1, tSwitchTime := longPressDelay);
fbKomoraVent(bOn := eib_vent_komora, bOff := NOT eib_vent_komora, bToggle := fbKomora1_sw.bLongClick);
eib_vent_komora := fbKomoraVent.bLight;
vent_komora := fbKomoraVent.bLight;
fbKomoraLight(button := fbKomora1_sw.bShortClick, duration := lightDuration, sensor := moove_komora, knx := eib_komora_l);
komora_l := fbKomoraLight.out;
eib_komora_l := fbKomoraLight.out;
fbSu1_1sw(bSwitch := sw_su1_1, tSwitchTime := longPressDelay);
fbSu1_l(bOn := eib_su1_l, bOff := NOT eib_su1_l, bToggle := sw_tambur_su XOR fbSu1_1sw.bShortClick);
su1_l := fbSu1_l.bLight;
eib_su1_l := fbSu1_l.bLight;
fbSu1Vent(bOn := eib_vent_su1, bOff := NOT eib_vent_su1, bToggle := fbSu1_1sw.bLongClick);
vent_su1 := fbSu1Vent.bLight;
eib_vent_su1 := fbSu1Vent.bLight;
fbSu1_rakovyna(bOn := eib_su1_rakovyna, bOff := NOT eib_su1_rakovyna, bToggle := sw_su1_2);
su1_rakovyna := fbSu1_rakovyna.bLight;
eib_su1_rakovyna := fbSu1_rakovyna.bLight;
fbKuh_su2_sw(bSwitch := sw_kuh_su2, tSwitchTime := longPressDelay);
fbSu2_l(bOn := eib_su2_l, bOff := NOT eib_su2_l, bToggle := fbKuh_su2_sw.bShortClick);
su2_l := fbSu2_l.bLight;
eib_su2_l := fbSu2_l.bLight;
fbSu2_dush(bOn := eib_su2_dush, bOff := NOT eib_su2_dush, bToggle := fbKuh_su2_sw.bLongClick);
su2_dush := fbSu2_dush.bLight;
su2_polytsi := fbSu2_dush.bLight;
eib_su2_dush := fbSu2_dush.bLight;
fbSu2_bra(bOn := eib_su2_bra, bOff := NOT eib_su2_bra);
su2_bra := fbSu2_bra.bLight;
eib_su2_bra := fbSu2_bra.bLight;
fbDush_sw(bSwitch := sw_su2, tSwitchTime := longPressDelay);
fbDush(bOn := eib_dush, bOff := NOT eib_dush, bToggle := fbDush_sw.bShortClick);
dush := fbDush.bLight;
eib_dush := fbDush.bLight;
fbDush_vent(bOn := eib_vent_dush, bOff := NOT eib_vent_dush, bToggle := fbDush_sw.bLongClick);
vent_dush := fbDush_vent.bLight;
eib_vent_dush := fbDush_vent.bLight;
fbKuh1_sw(bSwitch := sw_kuh1, tSwitchTime := longPressDelay);
fbKuhnya(bOn := eib_kuhnya1, bOff := NOT eib_kuhnya1, bToggle := fbKuh1_sw.bShortClick);
kuhnya1 := fbKuhnya.bLight;
kuhnya2 := fbKuhnya.bLight;
eib_kuhnya1 := fbKuhnya.bLight;
fbKuhnyaVent(bOn := eib_vent_kuh_low, bOff := NOT eib_vent_kuh_low, bToggle := fbKuh1_sw.bLongClick);
vent_kuh_low := fbKuhnyaVent.bLight;
eib_vent_kuh_low := fbKuhnyaVent.bLight;
fbSmugy(bOn := eib_vitalnya_smugy1, bOff := NOT eib_vitalnya_smugy1, bToggle := sw_vitalnya1 XOR sw_kuh2);
vitalnya_smugy1 := fbSmugy.bLight;
vitalnya_smugy2 := fbSmugy.bLight;
eib_vitalnya_smugy1 := fbSmugy.bLight;
fbVitalnya_l(bOn := eib_vitalnya_l, bOff := NOT eib_vitalnya_l, bToggle := sw_vitalnya2 XOR sw_kuh4);
vitalnya_l := fbVitalnya_l.bLight;
eib_vitalnya_l := fbVitalnya_l.bLight;
fbTerassa(bOn := eib_terassa, bOff := NOT eib_terassa, bToggle := sw_vitalnya3);
terassa := fbTerassa.bLight;
eib_terassa := fbTerassa.bLight;
fbProkladka(bOn := eib_vitalnya_prokladka, bOff := NOT eib_vitalnya_prokladka, bToggle := sw_kuh3);
vitalnya_prokladka := fbProkladka.bLight;
eib_vitalnya_prokladka := fbProkladka.bLight;
fbTerassa_stina(bOn := eib_terassa_stina, bOff := NOT eib_terassa_stina, bToggle := sw_vitalnya3);
terassa_stina := fbTerassa_stina.bLight;
eib_terassa_stina := fbTerassa_stina.bLight;
fbSkhody2Pov(bOn := eib_skhody2pov, bOff := NOT eib_skhody2pov, bToggle := sw_tambur1_2);
skhody2pov := fbSkhody2Pov.bLight;
eib_skhody2pov := fbSkhody2Pov.bLight;
fbTambur3_sw(bSwitch := sw_tambur3, tSwitchTime := longPressDelay);
fbPidval_shody(bOn := eib_pidval_shody, bOff := NOT eib_pidval_shody, bToggle := fbTambur3_sw.bShortClick);
pidval_shody := fbPidval_shody.bLight;
eib_pidval_shody := fbPidval_shody.bLight;
fbTamburLight(button := _t691, duration := lightDuration, sensor := _t520, knx := eib_tambur_l);
_t520 := MUX(BOOL_TO_INT(bDarkOutside), TRUE, moove_korydor);
_t691 := sw_tambur1 XOR sw_vhid1;
eib_tambur_l := fbTamburLight.out;
tambur_l := fbTamburLight.out;
END_PROGRAM

(* POU lights/fbMoovingSensorLight, ST *)
FUNCTION_BLOCK fbMoovingSensorLight
VAR_INPUT
	button:BOOL;
	duration:TIME;
	sensor:BOOL;
	knx:BOOL;
END_VAR
VAR_OUTPUT
	out: BOOL;
END_VAR
VAR
	fbStairwayLight_00			: FB_StairwellLight;
	button_rising				: R_TRIG;
	sensor_falling				: F_TRIG;
	timer_falling					: F_TRIG;
	knx_falling					: F_TRIG;
	knx_rising					: R_TRIG;
END_VAR

VAR_IN_OUT
END_VAR
knx_rising(CLK:=knx);
knx_falling(CLK:=knx);
button_rising(CLK:=button);
sensor_falling(CLK:= sensor);
timer_falling(clk:=fbStairwayLight_00.bStart);

IF sensor_falling.Q AND NOT out THEN
	fbStairwayLight_00.bOff:=FALSE;
END_IF

fbStairwayLight_00(
	bSwitch:=NOT sensor AND NOT out,
	tLightDuration:=duration,
	tPreWarningStart:=t#100s,
	tPreWarningDuration:=t#500ms);

IF fbStairwayLight_00.bStart THEN
	out := fbStairwayLight_00.bLight;
END_IF

IF timer_falling.Q THEN
	out:=FALSE;
END_IF




IF knx_rising.Q OR knx_falling.Q THEN
	out:= knx;
	IF knx_falling.Q THEN
		fbStairwayLight_00.bOff:=TRUE;
	END_IF
END_IF

IF button_rising.Q THEN
	out:= NOT out;
	fbStairwayLight_00.bOff:=TRUE;
END_IF
END_FUNCTION_BLOCK

(* POU heat, ST *)
PROGRAM heat
VAR
	temp_measure: TOF;
	t_vhid: REAL;
	t_dush: REAL;
	t_kuh: REAL;
	t_vhid_stina: REAL;

	t_max: SINT;
	t_min: SINT;
	t_out: REAL;
	i: INT;
	t_vhid_sum: REAL;
	t_dush_sum: REAL;
	t_vhid_stina_sum: REAL;
	t_kuh_sum: REAL;

	t_vhidPrev: REAL;
	t_dushPrev: REAL;
	t_vhid_stinaPrev: REAL;
	t_kuhPrev: REAL;

	delta_kuh: REAL;
	delta_vhid_stina: REAL;
	delta_dush: REAL;
	delta_vhid: REAL;
	retry:BOOL:=TRUE;(*переміряти температуру*)
	iRetryCounter: INT;
END_VAR
t_min:=0;
IF bT_out_sign THEN t_out:=0-t_out3; ELSE t_out:=t_out3; END_IF;

IF t_out >=17 AND skvazhyna THEN
	freecooling:=TRUE; (*freecooling means cold water in the system. There's hot water if it's FALSE*)
ELSE
	IF t_out<=12 THEN
		freecooling:=FALSE;
	END_IF
END_IF

	fancoil_vitalnya_low:=m_fancoil_vitalnya_low;
	fancoil_vitalnya_med:=m_fancoil_vitalnya_med;
	fancoil_vitalnya_high:=m_fancoil_vitalnya_high;
(*клапан управляється з 3го поверху*)


(*фільтр показань сенсорів температури*)
CASE i OF
0..500: init;
ELSE
	IF retry THEN
		temp_measure.PT:=t#2s;
	ELSE
		temp_measure.PT:=t#5m;
	END_IF
	IF retry THEN
		IF iRetryCounter >5 THEN iRetryCounter:=0; i:=0; ELSE iRetryCounter:=iRetryCounter+1; END_IF;
	END_IF;
	temp_measure( IN:=NOT temp_measure.q); (*перевіряти температуру кожні 20 хв*)

IF NOT temp_measure.Q THEN

	delta_kuh:=ABS(t_kuhPrev-temp_kuh*0.1);
	delta_vhid_stina:=ABS(t_vhid_stinaPrev-temp_vhid_stina*0.1);
	delta_dush:=ABS(t_dushPrev-temp_dush*0.1);
	delta_vhid:=ABS(t_vhidPrev-temp_vhid*0.1);
	retry:=FALSE;
	IF delta_kuh<1 THEN
		t_kuh:= temp_kuh * 0.1;
	ELSE
		t_kuh:=t_kuhPrev;
		retry:=TRUE;
	END_IF

	IF delta_vhid_stina<1 THEN
		t_vhid_stina:= temp_vhid_stina * 0.1;
	ELSE
		t_vhid_stina:=t_vhid_stinaPrev;
		retry:=TRUE;
	END_IF

	IF delta_dush<1 THEN
		t_dush:= temp_dush * 0.1;
	ELSE
		t_dush:=t_dushPrev;
		retry:=TRUE;
	END_IF

	IF delta_vhid<1 THEN
		t_vhid:= temp_vhid * 0.1;
	ELSE
		t_vhid:=t_vhidPrev;
		retry:=TRUE;
	END_IF

	t_kuhPrev:=t_kuh;
	t_vhid_stinaPrev:=t_vhid_stina;
	t_dushPrev:=t_dush;
	t_vhidPrev:=t_vhid;

END_IF
END_CASE

IF t_out>12 THEN
	t_max:=t_min;
ELSE
	IF t_out >0 THEN
		t_max:=10;
	ELSE
		t_max:=35;
	END_IF
END_IF

	IF t_vhid >=t_max THEN
		collector_vhid:=0;
	END_IF

	IF t_vhid <t_min THEN
		collector_vhid:=1;
	END_IF

	IF t_vhid_stina >=t_max THEN
		collector_vhid_stina:=0;
	END_IF

	IF t_vhid_stina <t_min THEN
		collector_vhid_stina:=1;
	END_IF

	IF t_dush >=t_max THEN
		collector_su2:=0;
	END_IF

	IF t_dush <t_min THEN
		collector_su2:=1;
	END_IF

	IF t_kuh<t_min THEN (*відкрити колектори, якщо підлога холодніша нижньої межі*)
		collector_vitalnya1:=1;
		collector_kuh:=1;
		collector_vitalnya2:=1;
	ELSE
		IF t_kuh >=t_max THEN (*закрити колектори, якщо підлога тепліша верхньої межі*)
			collector_vitalnya1:=0;
			collector_kuh:=0;
			collector_vitalnya2:=0;
			ELSE
				collector_vitalnya1:=tepla_pidloga;
				collector_kuh:=tepla_pidloga;
				collector_vitalnya2:=tepla_pidloga;
		END_IF
	END_IF
END_PROGRAM
ACTION init:
IF i=500 THEN
	t_vhidPrev:=t_vhid_sum/i;
	t_dushPrev:=t_dush_sum/i;
	t_vhid_stinaPrev:=t_vhid_stina_sum/i;
	t_kuhPrev:=t_kuh_sum/i;
	t_vhid_sum:=0;
	t_dush_sum:=0;
	t_vhid_stina_sum:=0;
	t_kuh_sum:=0;
	i:=501;
ELSE
	t_vhid_sum:=t_vhid_sum+temp_vhid*0.1;
	t_dush_sum:=t_dush_sum+temp_dush*0.1;
	t_vhid_stina_sum:=t_vhid_stina_sum+temp_vhid_stina*0.1;
	t_kuh_sum:=t_kuh_sum+temp_kuh*0.1;
	i:=i+1;
END_IF
END_ACTION

(* POU ADS_write, ST *)
PROGRAM ADS_write
VAR
	write_timeout: TIME;
	b_write3, b_write2: BOOL;
	write_ads3, write_ads2: ADSWRITE;

	timer3, timer2:TP;
	errorcounter3, errorcounter2, pack_c:CTU ;
	test_word: WORD;
	i,j,i1,j1: INT;
	data_changed: BOOL;
	try_again2, try_again3: BOOL;
	temp: INT;
	SENT2, SENT3:F_TRIG;
	SNT_CNT2, SNT_CNT3:CTU;
	fb_heartbeat_timer: TON;
END_VAR
data2floor[0].0:=sw_tambur1_2;
data2floor[0].1:=sw_vhid2;

data2floor[1].0:=moove_kino;
data2floor[1].1:=moove_skhody1_2;
data2floor[1].2:=moove_studio;
data2floor[1].3:=moove_kabinet;
data2floor[1].4:=Light.fbTambur3_sw.bLongClick;

data3floor[0].0:=moove_garderob;
data3floor[0].1:=moove_tambur3;
data3floor[0].2:=moove_dytjacha;
data3floor[0].3:=moove_spalnya;
data3floor[0].4:=moove_korydor3;
data3floor[0].5:=moove_skhody2_3;

data3floor[1].0:=komora_l;
data3floor[1].1:=su1_l;
data3floor[1].2:=topochna_l;
data3floor[1].3:=su2_bra	;
data3floor[1].4:=su2_l;
data3floor[1].5:=su1_rakovyna;
data3floor[1].6:=su2_dush;
data3floor[1].7:=dush;

data3floor[2].0:=kuhnya1	;
data3floor[2].1:=vitalnya_smugy1;
data3floor[2].2:=vitalnya_l;
data3floor[2].3:=vitalnya_prokladka;
data3floor[2].4:=terassa_stina	;
data3floor[2].5:=pidval_shody	;
data3floor[2].6:=terassa;
data3floor[2].7:=skhody2pov;

data3floor[3].4:=tambur_l;
data3floor[3].5:=vent_su1;
data3floor[3].6:=vent_kuh_low;
data3floor[3].7:=vent_dush;
data3floor[3].0:=vent_komora;
data3floor[3].1:=vent_kuh_high;



write_timeout:=t#1s;
fb_heartbeat_timer(in:=NOT fb_heartbeat_timer.Q, pt:=t#10s);

FOR i:=0 TO (SIZEOF(data2floor)-1)-1 DO
	IF data2floor[i]<>data2floor_prev[i] THEN
		b_write2:=TRUE;
		EXIT;
	ELSE
		b_write2:=FALSE;
	END_IF
END_FOR

IF try_again2 AND NOT timer2.Q THEN
	b_write2:=TRUE;
	try_again2:=FALSE;
END_IF


IF write_ads2.BUSY THEN b_write2:=FALSE; END_IF

	write_ads2(
		NETID:=ads_adr2,
		PORT:=800,
		IDXGRP:=16#4020,
		IDXOFFS:=100,
		WRITE:=b_write2,
		TMOUT:=write_timeout,
		LEN:=SIZEOF(data2floor),
		SRCADDR:=ADR(data2floor));

IF write_ads2.ERR AND NOT timer2.Q THEN
	timer2.IN:=TRUE;
	try_again2:=TRUE;
END_IF
timer2(PT:=write_timeout);
timer2.IN:=FALSE;

FOR j:=0 TO (SIZEOF(data2floor)-1)-1 DO
	data2floor_prev[j]:=data2floor[j];
END_FOR

SENT2(CLK:=write_ads2.BUSY);

IF NOT write_ads2.ERR THEN
	SNT_CNT2(CU:=SENT2.Q);
END_IF

(*3floor*)
FOR i1:=0 TO (SIZEOF(data3floor)-1)-1DO
	IF data3floor[i1]<>data3floor_prev[i1] OR fb_heartbeat_timer.Q  THEN
		b_write3:=TRUE;
		EXIT;
	ELSE
		b_write3:=FALSE;
	END_IF
END_FOR

IF try_again3 AND NOT timer3.Q THEN
	b_write3:=TRUE;
	try_again3:=FALSE;
END_IF


IF write_ads3.BUSY THEN b_write3:=FALSE; END_IF

	write_ads3(
		NETID:=ads_adr3,
		PORT:=801,
		IDXGRP:=16#4020,
		IDXOFFS:=100,
		WRITE:=b_write3,
		TMOUT:=write_timeout,
		LEN:=SIZEOF(data3floor),
		SRCADDR:=ADR(data3floor));

IF write_ads3.ERR AND NOT timer3.Q THEN
	timer3.IN:=TRUE;
	try_again3:=TRUE;
END_IF
timer3(PT:=write_timeout);
timer3.IN:=FALSE;

SENT3(CLK:=write_ads3.BUSY);

IF NOT write_ads3.ERR THEN
	SNT_CNT3(CU:=SENT3.Q);
END_IF

FOR j1:=0 TO (SIZEOF(data3floor)-1)-1 DO
	data3floor_prev[j1]:=data3floor[j1];
END_FOR
END_PROGRAM

(* POU lights/SWITCH, ST *)
FUNCTION_BLOCK SWITCH
VAR_INPUT
	IN:BOOL;
	SWITCH_DELAY:TIME; (*різниця між коротким і довгим натисненням*)
	SHORT_OFF_DELAY, LONG_OFF_DELAY: TIME; (*час затримки вимкнення по короткому та довгому натисненню*)
	MODE:STRING; (*delayed, light, light&vent, short&long, delayed_short&long, *)
	NUMBER_OF_OUTS:INT;
END_VAR
VAR_OUTPUT
	Q_SHORT:BOOL:=FALSE;
	Q_SHORT_D: BOOL;(*вихід для вимкнення із затримкою, вмикається разом із виходом короткого натискання*)
	Q_LONG:BOOL:=FALSE;
	Q_LONG_D:BOOL; (*вихід для вимкнення із затримкою, вмикається разом із виходом довгого натискання*)
END_VAR
VAR
	STAN:BOOL:=FALSE;
	Q_S_fall:F_TRIG; (*ловить задній фронт вихода короткого натискання*)
	Q_S_rise:F_TRIG; (*ловить задній фронт вихода короткого натискання*)
	Q_L_fall:F_TRIG;(*ловить задній фронт вихода довгого натискання*)
	chas: TIME; (*час доки кнопка натиснена*)

	long: BOOL; (*стає тру, якщо було довге натиснення*)
	short: BOOL; (*стає тру, якщо було коротке натиснення*)
	timer, short_off_delay_timer, long_off_delay_timer: TON; (*таймери: час натискання, час переключення відкладеного виходу по довгому та короткому натисканнях*)
	up: BOOL; (*кнопка натиснена*)

	delay_l, delay_s:BOOL; (*запускати таймери відкладеного вимкнення*)

	turn_off_long: BOOL;
	start_l, start_s:BOOL;
END_VAR
short:=0;
long:=0;
timer(IN:=IN AND STAN, PT:=t#10s);
IF IN AND STAN THEN
	chas:=timer.ET;
	up:=1;
ELSE
up:=0;
END_IF;

IF NOT IN AND NOT STAN THEN
chas:=t#0ms;
END_IF;

IF STAN AND NOT IN THEN
	IF chas <SWITCH_DELAY THEN
		short:=1;
		Q_SHORT:= NOT Q_SHORT;
	END_IF;
	IF chas>=SWITCH_DELAY THEN
		Q_LONG:= NOT Q_LONG;
		long:=1;
	END_IF;
END_IF;

(*затримка вимикання*)
Q_L_fall(CLK:=Q_LONG);
Q_S_fall(CLK:=Q_SHORT);
Q_S_rise(CLK:=Q_SHORT);

IF Q_L_FALL.Q THEN
		start_l:=TRUE;
END_IF

IF Q_S_FALL.Q THEN
	start_s:=TRUE;
END_IF

IF MODE='light&vent' THEN
	IF start_s THEN start_l:=start_s; END_IF
END_IF

IF LONG_OFF_DELAY <> t#0ms THEN (*виконувати лише якщо в блок переданий параметр затримки на вимкнення*)

	IF Q_LONG THEN
		Q_LONG_D:=Q_LONG;
	END_IF

	long_off_delay_timer(IN:=start_l, PT:=LONG_OFF_DELAY);

	IF long_off_delay_timer.Q THEN
		Q_LONG_D:=FALSE;
		start_l:=FALSE;
	END_IF

ELSE
	Q_LONG_D:=Q_LONG;
END_IF

IF SHORT_OFF_DELAY <> t#0ms THEN (*виконувати лише якщо в блок переданий параметр затримки на вимкнення*)

	IF Q_SHORT THEN
		Q_SHORT_D:=Q_SHORT;
	END_IF

	short_off_delay_timer(IN:=start_s, PT:=SHORT_OFF_DELAY);

	IF short_off_delay_timer.Q THEN
		Q_SHORT_D:=FALSE;
		start_s:=FALSE;
	END_IF


ELSE
	Q_SHORT_D:=Q_SHORT;
END_IF

IF MODE='delayed' THEN
	Q_LONG:=Q_LONG_D;
	Q_SHORT:=Q_SHORT_D;
END_IF
(*працють лише короткі замикання*)
IF MODE='light' THEN
	Q_SHORT_D:=FALSE;
	Q_LONG:=Q_SHORT;
	Q_LONG_D:=FALSE;
END_IF
(*затримки не працюють*)
IF MODE='short&long' THEN
	Q_SHORT_D:=FALSE;
	Q_LONG_D:=FALSE;
END_IF
(*при вимкненні всього світла вимикати вентилятор і затримкою*)
IF MODE='light&vent' THEN
	IF NOT Q_SHORT AND Q_LONG THEN
		Q_LONG:=Q_LONG_D;
	END_IF
END_IF

STAN := IN;
END_FUNCTION_BLOCK
